FUNCTION_BLOCK FB_PowerControlledHeaterFan EXTENDS FB_Actuator2Point

VAR
	
	//I/O Links	
	bSetStatusOn_OUT 	AT %Q*	: 	BOOL := FALSE;		
	
END_VAR

SelectControlMode();

METHOD SetState_BO : BOOL
VAR_INPUT
END_VAR
//output
bSetStatusOn_OUT := bSetStatusOn;
END_METHOD

END_FUNCTION_BLOCK

(* stored: Version 1.1.0.1, ProductVersion 3.1.4024.6
   POU FB_PowerControlledHeaterFan: Id {10dcde4f-7a77-4815-919a-97a9baa05130}, SpecialFunc None
   Method SetState_BO: Id {d8943a6b-21e0-4638-9af5-20b5899f0cc2} *)
